// TIA Portal V16 export
// export: Created 2023-08-28T09:37:43.5818194Z, ExportSetting WithDefaults, DisplayName Totally Integrated Automation Portal, DisplayVersion V16 Update 6, DisplayName TIA Portal Version Control Interface, DisplayVersion V16 Update 2, DisplayName TIA Portal Openness, DisplayVersion V16 Update 6, DisplayName STEP 7 Professional, DisplayVersion V16 Update 6, DisplayName STEP 7 Safety, DisplayVersion V16, DisplayName WinCC Advanced, DisplayVersion V16 Update 6
FUNCTION_BLOCK "04_A_Out_analog"   // FB23, LAD
TITLE = Output analogs
{ S7_Optimized_Access := 'TRUE' }
AUTHOR : rtecmer
VERSION : 0.1
// Obsługa wyjść analogowych
// stored: AutoNumber true, IsIECCheckEnabled false, IsRetainMemResEnabled false, MemoryReserve 100, SetENOAutomatically false, UDAEnableTagReadback false
   VAR
      Temp_SV_Int { ExternalAccessible := 'False'; ExternalVisible := 'False'; ExternalWritable := 'False'} : Int;
   END_VAR
   VAR_TEMP   // added for the SCL form of the ladder/FBD networks
      _w1 : Bool;
   END_VAR
BEGIN

REGION Network 1: Manual SV skalowanie
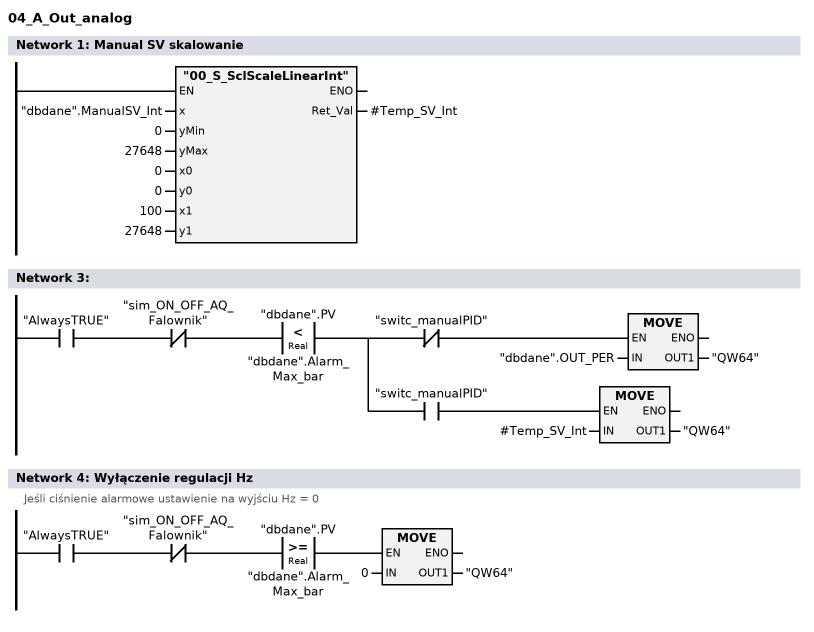
   RUNG wire#powerrail
      "00_S_SclScaleLinearInt"(x := "dbdane".ManualSV_Int, yMin := 0, yMax := 27648, x0 := 0, y0 := 0, x1 := 100, y1 := 27648, Ret_Val => #Temp_SV_Int)
   END_RUNG
   // the same network as SCL:
   #Temp_SV_Int := "00_S_SclScaleLinearInt"(x := "dbdane".ManualSV_Int,
                           yMin := 0,
                           yMax := 27648,
                           x0 := 0,
                           y0 := 0,
                           x1 := 100,
                           y1 := 27648);
END_REGION

REGION Network 3
   RUNG wire#powerrail
      Contact( "AlwaysTRUE" )
      I_Contact( "sim_ON_OFF_AQ_Falownik" )
      { S7_Templates := "SrcType := Real" } LT_Contact(in1 := "dbdane".PV, in2 := "dbdane".Alarm_Max_bar)
      wire#w1
      I_Contact( "switc_manualPID" )
      { S7_GenerateENO := "TRUE" } Move(in := "dbdane".OUT_PER, out1 => "QW64")
   END_RUNG
   RUNG wire#w1
      Contact( "switc_manualPID" )
      { S7_GenerateENO := "TRUE" } Move(in := #Temp_SV_Int, out1 => "QW64")
   END_RUNG
   // the same network as SCL:
   #_w1 := "AlwaysTRUE" AND NOT "sim_ON_OFF_AQ_Falownik" AND ("dbdane".PV < "dbdane".Alarm_Max_bar);
   IF #_w1 AND NOT "switc_manualPID" THEN "QW64" := "dbdane".OUT_PER; END_IF;
   IF #_w1 AND "switc_manualPID" THEN "QW64" := #Temp_SV_Int; END_IF;
END_REGION

REGION Network 4: Wyłączenie regulacji Hz
   // Jeśli ciśnienie alarmowe ustawienie na wyjściu Hz = 0
   RUNG wire#powerrail
      Contact( "AlwaysTRUE" )
      I_Contact( "sim_ON_OFF_AQ_Falownik" )
      { S7_Templates := "SrcType := Real" } GE_Contact(in1 := "dbdane".PV, in2 := "dbdane".Alarm_Max_bar)
      { S7_GenerateENO := "TRUE" } Move(in := 0, out1 => "QW64")
   END_RUNG
   // the same network as SCL:
   IF "AlwaysTRUE" AND NOT "sim_ON_OFF_AQ_Falownik" AND ("dbdane".PV >= "dbdane".Alarm_Max_bar) THEN
       "QW64" := 0;
   END_IF;
END_REGION
END_FUNCTION_BLOCK
